FUNCTION_BLOCK FB_TransferirPale_SFC

VAR_IN_OUT
	TpoCintaRetenedor: TIME;
    TpoPaleSalida: TIME;
    TpoPaleTransferencia: TIME;
END_VAR


VAR_INPUT
    // SFC-Flags
    SFCPause: BOOL;
    SFCReset: BOOL;
    
    // Indicadores de sincronizacion
    Ack: BOOL := TRUE;
    Execute: BOOL;
    
    // Entradas
    PresenciaPale: BOOL;
END_VAR
VAR_OUTPUT
    // Indicadores de sincronizacion
    Done: BOOL;
    Ready: BOOL;
    // Salidas
    CintaActiva: BOOL;
    RetenedorBaja: BOOL;
	SeparadorSube: BOOL;
END_VAR
VAR
END_VAR

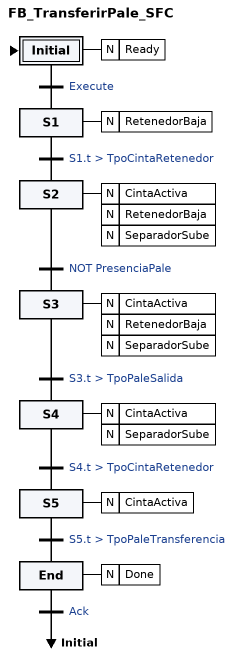
INITIAL_STEP Initial:
    Ready(N);
END_STEP
TRANSITION FROM Initial TO S1
    := Execute;
END_TRANSITION
STEP S1:
    RetenedorBaja(N);
END_STEP
TRANSITION FROM S1 TO S2
    := S1.t > TpoCintaRetenedor;
END_TRANSITION
STEP S2:
    CintaActiva(N);
    RetenedorBaja(N);
    SeparadorSube(N);
END_STEP
TRANSITION FROM S2 TO S3
    := NOT PresenciaPale;
END_TRANSITION
STEP S3:
    CintaActiva(N);
    RetenedorBaja(N);
    SeparadorSube(N);
END_STEP
TRANSITION FROM S3 TO S4
    := S3.t > TpoPaleSalida;
END_TRANSITION
STEP S4:
    CintaActiva(N);
    SeparadorSube(N);
END_STEP
TRANSITION FROM S4 TO S5
    := S4.t > TpoCintaRetenedor;
END_TRANSITION
STEP S5:
    CintaActiva(N);
END_STEP
TRANSITION FROM S5 TO End
    := S5.t > TpoPaleTransferencia;
END_TRANSITION
STEP End:
    Done(N);
END_STEP
TRANSITION FROM End TO Initial
    := Ack;
END_TRANSITION

END_FUNCTION_BLOCK

(* stored: Version 1.1.0.1, ProductVersion 3.1.4024.9
   POU FB_TransferirPale_SFC: Id {294b1446-deed-4479-9db5-1759d0b39862}, SpecialFunc None *)
